FUNCTION_BLOCK E_CTU (* Event driven up counter *)
  (* Standard: 61499-1 Annex 2; Description: Copyright (c) 2017 fortiss GmbH This program and the accompanying materials are made available under the terms of the Eclipse Public License 2.0 which is available at https://www.eclipse.org/legal/epl-2.0/ SPDX-License-Identifier: EPL-2.0 *)
  (* Version 1.0, 2017-09-21, Alois Zoitl, fortiss GmbH, initial API and implementation and/or initial documentation *)
  (* Version 3.0, 2025-04-14, Patrick Aigner, changed package *)
  PACKAGE iec61499::events;
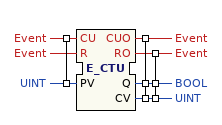
  EVENT_INPUT
    CU WITH PV; (* Count up *)
    R; (* Reset *)
  END_EVENT
  EVENT_OUTPUT
    CUO WITH Q, CV; (* Count up output *)
    RO WITH Q, CV; (* Reset output *)
  END_EVENT
  VAR_INPUT
    PV : UINT; (* Process Value *)
  END_VAR
  VAR_OUTPUT
    Q : BOOL; (* True if CV >= PV *)
    CV : UINT; (* Counter Value *)
  END_VAR
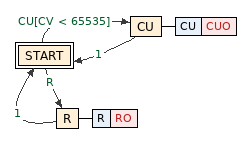
  EC_STATES
    START; (* Initial State *)
    CU : CU -> CUO; (* Count Up *)
    R : R -> RO; (* Reset *)
  END_STATES
  EC_TRANSITIONS
    START TO CU := CU[CV < 65535];
    CU TO START := 1;
    START TO R := R;
    R TO START := 1;
  END_TRANSITIONS
  ALGORITHM R IN ST: (* reset counter *)
CV := 0;
Q := FALSE;
  END_ALGORITHM
  ALGORITHM CU IN ST: (* count up *)
CV := CV + 1;
Q  := (CV >= PV);
  END_ALGORITHM
END_FUNCTION_BLOCK
